// TIA Portal V18 export
VAR_GLOBAL   // PLC tag table "Default tag table"
   "mz encoder a" AT %I0.0 : Bool;
   "mz encoder b" AT %I0.1 : Bool;
   "my encoder a" AT %I0.2 : Bool;
   "my encoder b" AT %I0.3 : Bool;
   "mx encoder a" AT %I0.4 : Bool;
   "mx encoder b" AT %I0.5 : Bool;
   "mz up indNOK" AT %I0.6 : Bool;
   "mz down indNOK" AT %I0.7 : Bool;
   "my fwd indNOK" AT %I1.0 : Bool;
   "my rev indNOK" AT %I1.1 : Bool;
   "mx right indNOK" AT %I1.2 : Bool;
   "mx left indNOK" AT %I1.3 : Bool;
   "mo1 tilt fwd indNOK" AT %I1.4 : Bool;
   "mo1 tilt rev indNOK" AT %I1.5 : Bool;
   "na(3)" AT %I1.6 : Bool;
   "na(4)" AT %I1.7 : Bool;
   ai_reserve AT %IW100 : Int;
   "ai_reserve(1)" AT %IW102 : Int;
   hscрезерв AT %ID812 : DInt;
   "hscрезерв(1)" AT %ID816 : DInt;
   "hscрезерв(2)" AT %ID820 : DInt;
   "mz hsc" AT %ID800 : DInt;
   "my hsc" AT %ID804 : DInt;
   "mx hsc" AT %ID808 : DInt;
   "a1_com_di50.0" AT %I50.0 : Bool;
   "a1_com_di50.1" AT %I50.1 : Bool;
   "a1_com_di50.2" AT %I50.2 : Bool;
   "a1_com_di50.3" AT %I50.3 : Bool;
   "a1_com_di50.4" AT %I50.4 : Bool;
   "a1_com_di50.5" AT %I50.5 : Bool;
   "a1_com_di50.6" AT %I50.6 : Bool;
   "a1_com_di50.7" AT %I50.7 : Bool;
   a1_com_di_byte AT %IB50 : Byte;
   "mo1 enc a" AT %I2.0 : Bool;
   "mo1 enc b" AT %I2.1 : Bool;
   "mo2 enc a" AT %I2.2 : Bool;
   "mo2 enc b" AT %I2.3 : Bool;
   "door enc a" AT %I2.4 : Bool;
   "door enc b" AT %I2.5 : Bool;
   "door closed 1 ind NOT" AT %I2.6 : Bool;
   "door open NOK 1 ind" AT %I2.7 : Bool;
   "res i" AT %I3.0 : Bool;
   "mo2 rot home ind" AT %I3.1 : Bool;
   "res i(1)" AT %I3.2 : Bool;
   "air pres ok" AT %I3.3 : Bool;
   "door closed 1 mech Excluded For Xray" AT %I3.4 : Bool;
   "door open 1 mech" AT %I3.5 : Bool;
   "na(1)" AT %I3.6 : Bool;
   "na(2)" AT %I3.7 : Bool;
   "ai_reserve(2)" AT %IW110 : Int;
   "ai_reserve(3)" AT %IW112 : Int;
   "hscрезерв(3)" AT %ID862 : DInt;
   "hscрезерв(4)" AT %ID866 : DInt;
   "hscрезерв(5)" AT %ID870 : DInt;
   "mo1 hsc" AT %ID850 : DInt;
   "mo2 hsc" AT %ID854 : DInt;
   "door hsc" AT %ID858 : DInt;
   "mz up mech" AT %I4.0 : Bool;
   "mz down mech" AT %I4.1 : Bool;
   "CAB phase check OK" AT %I4.2 : Bool;
   lightBarrierOK AT %I4.3 : Bool;
   "my fwd mech" AT %I4.4 : Bool;
   "my rev mech" AT %I4.5 : Bool;
   "xray coler ok" AT %I4.6 : Bool;
   ESTOP_AND_KEY_OK AT %I4.7 : Bool;
   "mx right mech" AT %I5.0 : Bool;
   "mx left mech" AT %I5.1 : Bool;
   "door closed 2 mech Excluded For Xray" AT %I5.2 : Bool;
   "door open 2 mech" AT %I5.3 : Bool;
   "mo1 tilt fwd mech" AT %I5.4 : Bool;
   "mo1 tilt rev mech" AT %I5.5 : Bool;
   "door closed 2 ind NOT" AT %I5.6 : Bool;
   "door open 2 ind NOT" AT %I5.7 : Bool;
   "desk door b close" AT %I6.0 : Bool;
   "desk door b open" AT %I6.1 : Bool;
   "desk o1 tilt b cw" AT %I6.2 : Bool;
   "desk o1 tilt b ccw" AT %I6.3 : Bool;
   "desk b home" AT %I6.4 : Bool;
   "desk b load unload" AT %I6.5 : Bool;
   "desk b laser centr" AT %I6.6 : Bool;
   "res i(3)" AT %I7.0 : Bool;
   "res i(4)" AT %I7.1 : Bool;
   ESTOP_OK AT %I7.2 : Bool;
   Y2_home_esw AT %I7.3 : Bool;
   "shutter open ind" AT %I7.5 : Bool;
   "shutter closed ind" AT %I7.4 : Bool;
   "ESTOP xray OK" AT %I7.6 : Bool;
   "res i(8)" AT %I7.7 : Bool;
   "detector safety ok" AT %I8.0 : Bool;
   "desk o2 rot b fwd" AT %I8.1 : Bool;
   "desk o2 rot b reverse" AT %I8.3 : Bool;
   "desk o2 rot b home" AT %I8.2 : Bool;
   "desk y  b rev" AT %I8.4 : Bool;
   "desk y b fwd" AT %I8.5 : Bool;
   "desk b defect next" AT %I8.6 : Bool;
   "desk b defect prev" AT %I8.7 : Bool;
   "desk sw manual" AT %I9.0 : Bool;
   "desk sw auto" AT %I9.1 : Bool;
   "desk b auto start" AT %I9.2 : Bool;
   "desk b defect mark" AT %I9.3 : Bool;
   "desk x b left" AT %I9.4 : Bool;
   "desk x b right" AT %I9.5 : Bool;
   "desk z up" AT %I9.7 : Bool;
   "desk z down" AT %I9.6 : Bool;
   "remote key activated" AT %I6.7 : Bool;
   "mz up" AT %Q0.1 : Bool;
   "mz down" AT %Q0.2 : Bool;
   "mz up STOP" AT %Q0.3 : Bool;
   "mz down STOP" AT %Q0.4 : Bool;
   "my fwd" AT %Q0.6 : Bool;
   "my rev" AT %Q0.5 : Bool;
   "my fwd STOP" AT %Q0.7 : Bool;
   "my rev STOP" AT %Q1.0 : Bool;
   "shutter out1.1" AT %Q1.1 : Bool;
   "na(5)" AT %Q1.2 : Bool;
   "na(6)" AT %Q1.3 : Bool;
   "na(7)" AT %Q1.4 : Bool;
   "na(8)" AT %Q1.5 : Bool;
   "na(9)" AT %Q1.6 : Bool;
   "na(10)" AT %Q1.7 : Bool;
   "mz up down speed" AT %QW100 : Int;
   "my fwd rev speed" AT %QW102 : Int;
   "a1_com_dq50.0" AT %Q50.0 : Bool;
   "a1_com_dq50.1" AT %Q50.1 : Bool;
   "a1_com_dq50.2" AT %Q50.2 : Bool;
   "a1_com_dq50.3" AT %Q50.3 : Bool;
   "a1_com_dq50.4" AT %Q50.4 : Bool;
   "a1_com_dq50.5" AT %Q50.5 : Bool;
   "a1_com_dq50.6" AT %Q50.6 : Bool;
   "a1_com_dq50.7" AT %Q50.7 : Bool;
   a1_com_dq_byte AT %QB50 : Byte;
   "column yellow" AT %Q2.0 : Bool;
   "column green" AT %Q2.1 : Bool;
   "column red" AT %Q2.2 : Bool;
   "detector power" AT %Q2.3 : Bool;
   "mx right" AT %Q2.5 : Bool;
   "mx left" AT %Q2.6 : Bool;
   "mx right STOP" AT %Q2.7 : Bool;
   "mx left STOP" AT %Q3.0 : Bool;
   "light barrier power" AT %Q3.1 : Bool;
   "res q" AT %Q2.4 : Bool;
   na AT %Q3.2 : Bool;
   na_1 AT %Q3.3 : Bool;
   na_2 AT %Q3.4 : Bool;
   na_3 AT %Q3.5 : Bool;
   na_4 AT %Q3.6 : Bool;
   na_5 AT %Q3.7 : Bool;
   "mx speed right left" AT %QW110 : Int;
   "mo1 tilt speed" AT %QW112 : Int;
   "mo1 tilt fwd" AT %Q4.1 : Bool;
   "mo1 tilt rev" AT %Q4.0 : Bool;
   "mo1 tilt fwd STOP" AT %Q4.2 : Bool;
   "mo1 tilt rev STOP" AT %Q4.3 : Bool;
   "mo2 rot cw" AT %Q4.4 : Bool;
   "mo2 rot ccw" AT %Q4.5 : Bool;
   "mo2 rot cw STOP" AT %Q4.6 : Bool;
   "mo2 rot ccw STOP" AT %Q4.7 : Bool;
   "door close" AT %Q5.0 : Bool;
   "door open" AT %Q5.1 : Bool;
   "door close STOP" AT %Q5.2 : Bool;
   "door open STOP" AT %Q5.3 : Bool;
   "magnet energize" AT %Q5.4 : Bool;
   "laser center energize" AT %Q5.5 : Bool;
   reserve_aq AT %QW118 : Int;
   "reserve_aq(1)" AT %QW120 : Int;
   "mo2 speed" AT %QW114 : Int;
   "door speed" AT %QW116 : Int;
   "desk siren finished" AT %Q6.1 : Bool;
   "desk siren error" AT %Q6.2 : Bool;
   "desk led auto on" AT %Q6.3 : Bool;
   "desk led shutter closed" AT %Q6.4 : Bool;
   "res q(1)" AT %Q6.0 : Bool;
   "remote power supNA" AT %Q6.5 : Bool;
   "res q(2)" AT %Q6.6 : Bool;
   "res q(3)" AT %Q6.7 : Bool;
   "res q(4)" AT %Q7.0 : Bool;
   "res q(5)" AT %Q7.1 : Bool;
   "res q(6)" AT %Q7.2 : Bool;
   "res q(7)" AT %Q7.3 : Bool;
   "res q(8)" AT %Q7.4 : Bool;
   "res q(9)" AT %Q7.5 : Bool;
   "res q(10)" AT %Q7.6 : Bool;
   "res q(11)77" AT %Q7.7 : Bool;
   erCOM_A1 AT %M0.0 : Bool;
   "erCOM_A1(1)" AT %M0.1 : Bool;
   wnDelay AT %M0.2 : Bool;
   MD_CYCLE AT %M0.3 : Bool;
END_VAR
VAR_GLOBAL CONSTANT   // user constants
   "None(1)" : Pip := 65535;
   "Automatic update(1)" : Pip := 0;
   "PIP 1(1)" : Pip := 1;
   "PIP 2(1)" : Pip := 2;
   "PIP 3(1)" : Pip := 3;
   "PIP 4(1)" : Pip := 4;
   "PIP OB Servo(1)" : Pip := 32768;
   "Local~MC(1)" : Hw_SubModule := 51;
   "Local~Exec(1)" : Hw_SubModule := 52;
   "Local(1)" : Hw_SubModule := 49;
   "Local~PROFINET_interface_1(1)" : Hw_Interface := 64;
   "Local~PROFINET_interface_1~Port_1(1)" : Hw_Interface := 65;
   "Local~PROFINET_interface_1~Port_2(1)" : Hw_Interface := 66;
   "Local~HSC_1(1)" : Hw_Hsc := 257;
   "Local~HSC_2(1)" : Hw_Hsc := 258;
   "Local~HSC_3(1)" : Hw_Hsc := 259;
   "Local~HSC_4(1)" : Hw_Hsc := 260;
   "Local~HSC_5(1)" : Hw_Hsc := 261;
   "Local~HSC_6(1)" : Hw_Hsc := 262;
   "Local~AI_2_AQ_2_1(1)" : Hw_SubModule := 263;
   "Local~DI_14_DQ_10_1(1)" : Hw_SubModule := 264;
   "Local~OPC_UA(1)" : Hw_SubModule := 117;
   "Local~Pulse_1(1)" : Hw_Pwm := 265;
   "Local~Pulse_2(1)" : Hw_Pwm := 266;
   "Local~Pulse_3(1)" : Hw_Pwm := 267;
   "Local~Pulse_4(1)" : Hw_Pwm := 268;
   "OB_Main(1)" : OB_PCYCLE := 1;
   "Local~A3_DI_16x24VDC_DQ_16xRelay_1" : Hw_SubModule := 269;
   "Local~A4_AQ_4x14BIT_1" : Hw_SubModule := 270;
   "Local~A5_DI_16x24VDC_DQ_16xRelay_2" : Hw_SubModule := 271;
   "Local~A6_DI_16x24VDC_1" : Hw_SubModule := 272;
   "Local~PROFINET_IO-System(1)" : Hw_IoSystem := 273;
   "A1_slave~PROFINET_interface_1~IODevice(1)" : Hw_Device := 275;
   "A1_slave~PROFINET_interface_1~bool0(1)" : Hw_SubModule := 277;
   "A1_slave~PROFINET_interface_1~bool1(1)" : Hw_SubModule := 278;
   "A1_slave~PROFINET_interface_1~analog0(1)" : Hw_SubModule := 279;
   "A1_slave~PROFINET_interface_1~anolog1(1)" : Hw_SubModule := 280;
   "A1_slave~PROFINET_interface_1~hsc(1)" : Hw_SubModule := 281;
   "A1_slave~PROFINET_interface_1~pulse(1)" : Hw_SubModule := 282;
   "A1_slave~PROFINET_interface_1~comm0(1)" : Hw_SubModule := 283;
   "A1_slave~PROFINET_interface_1~comm1" : Hw_SubModule := 284;
   "Local~Common(1)" : Hw_SubModule := 50;
   "Local~Device(1)" : Hw_Device := 32;
   "Local~Configuration(1)" : Hw_SubModule := 33;
   "OB_Cyclic interrupt" : OB_Cyclic := 30;
END_VAR
